FUNCTION_BLOCK CSWI (* Composite Function Block Type *)
  (* Standard: 61499-2 *)
  (* Version 0.0, 12/11/2023, Cheyan, Schneider Electric, template *)
  PACKAGE Main;
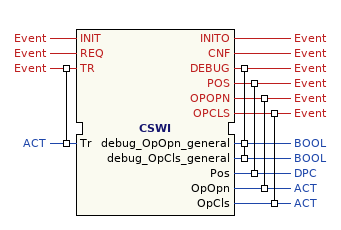
  EVENT_INPUT
    INIT; (* Initialization Request *)
    REQ; (* Normal Execution Request *)
    TR WITH Tr;
  END_EVENT
  EVENT_OUTPUT
    INITO; (* Initialization Confirm *)
    CNF; (* Execution Confirmation *)
    DEBUG WITH debug_OpOpn_general, debug_OpCls_general;
    POS WITH Pos;
    OPOPN WITH OpOpn;
    OPCLS WITH OpCls;
  END_EVENT
  VAR_INPUT
    Tr : ACT; (* Input event qualifier *)
  END_VAR
  VAR_OUTPUT
    debug_OpOpn_general : BOOL;
    debug_OpCls_general : BOOL;
    Pos : DPC;
    OpOpn : ACT;
    OpCls : ACT;
  END_VAR
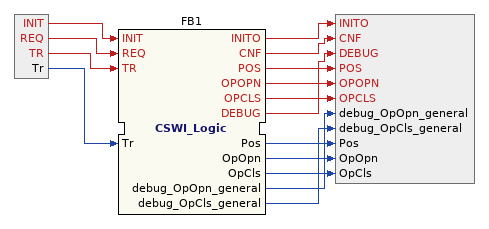
  FBS
    FB1 : CSWI_Logic;
  END_FBS
  EVENT_CONNECTIONS
    INIT TO FB1.INIT;
    REQ TO FB1.REQ;
    FB1.INITO TO INITO;
    FB1.CNF TO CNF;
    FB1.DEBUG TO DEBUG;
    TR TO FB1.TR;
    FB1.POS TO POS;
    FB1.OPOPN TO OPOPN;
    FB1.OPCLS TO OPCLS;
  END_CONNECTIONS
  DATA_CONNECTIONS
    FB1.debug_OpOpn_general TO debug_OpOpn_general;
    FB1.debug_OpCls_general TO debug_OpCls_general;
    Tr TO FB1.Tr;
    FB1.Pos TO Pos;
    FB1.OpOpn TO OpOpn;
    FB1.OpCls TO OpCls;
  END_CONNECTIONS
END_FUNCTION_BLOCK
